TYPE ST_DIS_Diagnosis :
STRUCT
	Chanel_0	: ST_DIS_Chanel_Diagnosis ;
	Chanel_1	: ST_DIS_Chanel_Diagnosis ;
	Chanel_2	: ST_DIS_Chanel_Diagnosis ;
	Chanel_3	: ST_DIS_Chanel_Diagnosis ;
	Chanel_4	: ST_DIS_Chanel_Diagnosis ;
	Chanel_5	: ST_DIS_Chanel_Diagnosis ;
	Chanel_6	: ST_DIS_Chanel_Diagnosis ;
	Chanel_7	: ST_DIS_Chanel_Diagnosis ;
END_STRUCT
END_TYPE

(* stored: Version 1.1.0.1
   DUT ST_DIS_Diagnosis: Id {43fdaa55-2e59-4bc0-9333-9e4ad9826933} *)
